FUNCTION TryConvert_DINT_TO_REAL : BOOL
VAR_INPUT
	in : DINT;
	out : REFERENCE TO REAL;
END_VAR

out := DINT_TO_REAL(in);
TryConvert_DINT_TO_REAL := TRUE;

END_FUNCTION

(* stored: Version 1.1.0.1, ProductVersion 3.1.4024.12
   POU TryConvert_DINT_TO_REAL: Id {c2d871c2-6211-4d4a-bccf-c62be106bf78}, SpecialFunc None *)
